(* PLC project  *)

CONFIGURATION SoftMotion General Axis Pool
END_CONFIGURATION
